FUNCTION_BLOCK FB_FileSaveAs_V02
VAR_INPUT
	i_bExecute					:BOOL;
	i_sSourcePath				:STRING;
	i_sDestinationPath			:STRING;
	i_sFileSourceName			:STRING;
	i_sFileDestName				:STRING;
END_VAR
VAR_OUTPUT
	q_bBusy						:BOOL;
	q_bDone						:BOOL;
	q_bError					:BOOL;
	q_sError					:STRING;
END_VAR
VAR
	fbSourceOpen				:FB_FileOpen;
	fbDestinationOpen			:FB_FileOpen;
	
	fbSourceRead				:FB_FileRead;
	fbDestinationWrite			:FB_FileWrite;
	
	fbSourceClose				:FB_FileClose;
	fbDestinationClose			:FB_FileClose;
	
	sSourceOpen					:STRING[300];
	sDestinationOpen			:STRING[300];

	arrData						:ARRAY[0..9999] OF BYTE;
	
	bOpen						:BOOL;
	bRead						:BOOL;
	bWrite						:BOOL;
	bClose						:BOOL;
	
	iStep						:INT;
END_VAR


CASE iStep OF
	
	0:
		q_bBusy:=FALSE;
		IF i_bExecute THEN
			q_sError:='';
			q_bError:=FALSE;
			q_bDone:=FALSE;
			q_bBusy:=TRUE;
			MEMSET(ADR(arrData),0,SIZEOF(arrData));
			iStep:=10;
		END_IF

	10:
		sSourceOpen := CONCAT(i_sSourcePath,i_sFileSourceName);
		sDestinationOpen := CONCAT(i_sDestinationPath,i_sFileDestName);
		iStep:=20;
		
	20:
		bOpen:=TRUE;
		IF NOT fbSourceOpen.bBusy AND NOT fbDestinationOpen.bBusy AND NOT fbSourceOpen.bError AND NOT fbDestinationOpen.bError THEN
			iStep:=30;
		ELSIF fbSourceOpen.bError OR fbDestinationOpen.bError THEN
			q_bError:=TRUE;
			q_sError:='Error opening files';
			iStep:=50;
		END_IF
		
	30:
		bRead:=TRUE;
		IF fbSourceRead.bBusy THEN
			iStep:=35;
		END_IF
	35:
		
		IF NOT fbSourceRead.bBusy AND NOT fbSourceRead.bError THEN
			iStep:=40;
		ELSIF fbSourceRead.bError THEN
			q_bError:=TRUE;
			q_sError:='Error reading source file';
			iStep:=50;
		END_IF
		
	40:
		bWrite:=TRUE;
		IF fbDestinationWrite.bBusy THEN
			iStep:=45;
		END_IF
	45:
		IF NOT fbDestinationWrite.bBusy AND NOT fbDestinationWrite.bError THEN
			iStep:=50;
		ELSIF fbDestinationWrite.bError THEN
			q_bError:=TRUE;
			q_sError:='Error writing source file';
			iStep:=50;
		END_IF
	50:
		bClose:=TRUE;
		IF NOT fbSourceClose.bBusy AND NOT fbDestinationClose.bBusy AND NOT fbSourceClose.bError AND NOT fbDestinationClose.bError THEN
			iStep:=100;
		ELSIF fbSourceClose.bError OR fbDestinationClose.bError THEN
			q_bError:=TRUE;
			q_sError:='Error closing files';
			iStep:=0;
		END_IF
		
	100:
		q_bDone:=TRUE;
		iStep:=0;
	
END_CASE

Cmd();

ACTION Cmd:
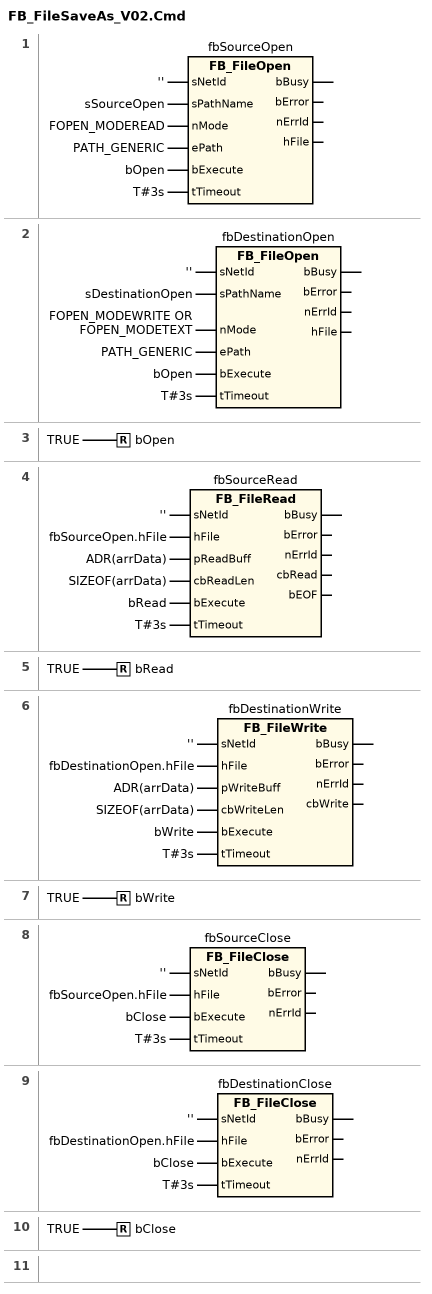
// NETWORK 1
fbSourceOpen(
    sNetId := '',
    sPathName := sSourceOpen,
    nMode := FOPEN_MODEREAD,
    ePath := PATH_GENERIC,
    bExecute := bOpen,
    tTimeout := T#3s); // FB_FileOpen

// NETWORK 2
fbDestinationOpen(
    sNetId := '',
    sPathName := sDestinationOpen,
    nMode := FOPEN_MODEWRITE OR FOPEN_MODETEXT,
    ePath := PATH_GENERIC,
    bExecute := bOpen,
    tTimeout := T#3s); // FB_FileOpen

// NETWORK 3
bOpen R= TRUE;

// NETWORK 4
fbSourceRead(
    sNetId := '',
    hFile := fbSourceOpen.hFile,
    pReadBuff := ADR(arrData),
    cbReadLen := SIZEOF(arrData),
    bExecute := bRead,
    tTimeout := T#3s); // FB_FileRead

// NETWORK 5
bRead R= TRUE;

// NETWORK 6
fbDestinationWrite(
    sNetId := '',
    hFile := fbDestinationOpen.hFile,
    pWriteBuff := ADR(arrData),
    cbWriteLen := SIZEOF(arrData),
    bExecute := bWrite,
    tTimeout := T#3s); // FB_FileWrite

// NETWORK 7
bWrite R= TRUE;

// NETWORK 8
fbSourceClose(sNetId := '', hFile := fbSourceOpen.hFile, bExecute := bClose, tTimeout := T#3s); // FB_FileClose

// NETWORK 9
fbDestinationClose(sNetId := '', hFile := fbDestinationOpen.hFile, bExecute := bClose, tTimeout := T#3s); // FB_FileClose

// NETWORK 10
bClose R= TRUE;

// NETWORK 11
END_ACTION

END_FUNCTION_BLOCK

(* stored: Version 1.1.0.1, ProductVersion 3.1.4024.12
   POU FB_FileSaveAs_V02: Id {e7a37c5f-b93c-47ca-89f9-01ab66e9a3a5}, SpecialFunc None
   Action Cmd: Id {3bc4d9e5-fcbf-4404-a471-ef99e0b49e99} *)
